FUNCTION_BLOCK TEST_MIN (* Test IEC 61131 MIN functions *)
  (* Standard: 61499-1 *)
  (* Version 0.0, 2006-09-12, JHC, Holobloc Inc *)
  (* Compiler header: package fb.rt.test; *)
  (* Compiler classdef: public class Simple extends SimpleFB *)
  (* Compiler Java Sun JDK 1.5.0 *)
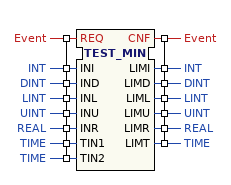
  EVENT_INPUT
    REQ WITH INI, INR, IND, INL, TIN1, INU, TIN2; (* Normal Execution Request *)
  END_EVENT
  EVENT_OUTPUT
    CNF WITH LIMI, LIMR, LIMD, LIML, LIMT, LIMU; (* Execution Confirmation *)
  END_EVENT
  VAR_INPUT
    INI : INT;
    IND : DINT;
    INL : LINT;
    INU : UINT;
    INR : REAL;
    TIN1 : TIME;
    TIN2 : TIME;
  END_VAR
  VAR_OUTPUT
    LIMI : INT; (* Output event qualifier *)
    LIMD : DINT;
    LIML : LINT;
    LIMU : UINT;
    LIMR : REAL;
    LIMT : TIME;
  END_VAR
  ALGORITHM REQ IN FBD: (* Normally executed algorithm *)
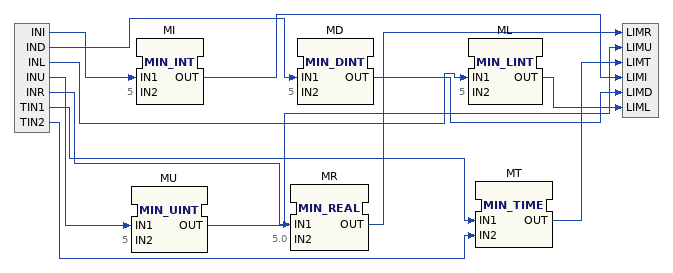
    FBS
      MI : MIN_INT(IN2 := 5);
      MR : MIN_REAL(IN2 := 5.0);
      ML : MIN_LINT(IN2 := 5);
      MT : MIN_TIME;
      MU : MIN_UINT(IN2 := 5);
      MD : MIN_DINT(IN2 := 5);
    END_FBS
    DATA_CONNECTIONS
      MR.OUT TO LIMR;
      MU.OUT TO LIMU;
      MT.OUT TO LIMT;
      INI TO MI.IN1;
      MI.OUT TO LIMI;
      IND TO MD.IN1;
      MD.OUT TO LIMD;
      INL TO ML.IN1;
      ML.OUT TO LIML;
      INU TO MU.IN1;
      INR TO MR.IN1;
      TIN1 TO MT.IN1;
      TIN2 TO MT.IN2;
    END_CONNECTIONS
  END_ALGORITHM
END_FUNCTION_BLOCK
